# EPICS autosave request: TC/iocBoot/iocTC-IOC-02/TC_02_settings.req
file "TC_02_built_settings.req"
